// Implicitly generated code : DO NOT EDIT
FUNCTION CheckRangeSigned : DINT
VAR_INPUT
	value, lower, upper: DINT;
END_VAR

// Implicitly generated code : Only an Implementation suggestion
IF (value < lower) THEN
	CheckRangeSigned := lower;
	gvlChecks.dCheckRangeSigned := gvlChecks.dCheckRangeSigned + 1;
ELSIF(value > upper) THEN
	CheckRangeSigned := upper;
	gvlChecks.dCheckRangeSigned := gvlChecks.dCheckRangeSigned + 1;
ELSE
	CheckRangeSigned := value;
END_IF

END_FUNCTION

(* stored: Version 1.1.0.1, ProductVersion 3.1.4026.13, FileIdentifier 06bb6c89f536b44a1d1363f2f79186121524c08d, FileSignature a3679237c02ce04c2389a63abbfb5ba8ff60ee3e0cdd669e226ea98376b7a9fbd910495cf2bae0008455ff6f149a71699004028c242f90576caee2a6d8c95a8e5e09f0c837d32ee51ccf47fb98d0d9f44c08d6f555fd5e55302d745704e7dc60723393b0a04a249b3d6376dc8e97e81bd85c9bb65dd02f611e5b12d7bf1734e43ef08af4955c648b7b77d60cfb9b8ea55517722aad7e1437e9c792ed4c99c06a01e5ee00c68dec4036a6fc6c43f0e74288835ead17a99e0574023ea136c6862e77a6a9127da16229e91593eb214565ee83f1d9b0a40835cc36129c4287f7faa131e4b9733a2a002ff3e3064c336d906cce6bb77b0e6c5fa4330cd3a43950916e
   POU CheckRangeSigned: Id {3f665f5c-f2d8-4cce-8287-4400ac7ad20d}, SpecialFunc CheckRangeSigned *)
